(* PLC project Standard Funtion Blocks, Beremiz Additional Function Blocks Library 1.0, author Laurent Bessard *)
(* stored: creationDateTime 2013-09-09T09:56:11, modificationDateTime 2013-09-10T22:45:31 *)

(* pluse out *)
FUNCTION_BLOCK StepperDriver
  VAR_INPUT
    CH : USINT;  (* 输出通道,范围由控制器决定,1-n *)
    MaxSpeed : UDINT;  (* 设定最高速度,单位Hz *)
    Acceleration : UDINT;  (* 设定最高加减速,单位Hz *)
    StepPinPolarity : BOOL;  (* 脉冲输出极性设定 *)
    DirectionPolarity : BOOL;  (* 方向输出极性设定 *)
    TargetAbs : DINT;  (* 绝对目标位置设定 *)
    TargetRel : DINT;  (* 相对目标位置设定 *)
    TargetSet : USINT;  (* 目标位置设定,1=绝对位置,2=相对位置,其它=不修改 *)
    Position : DINT;  (* 当前位置设定 *)
    PositionSet : BOOL;  (* 当前位置设定,1有效 *)
    Run : BOOL;  (* 1=运行,0=停止 *)
  END_VAR
  VAR_OUTPUT
    Running : BOOL;  (* 运行状态,1=正在运行,0=停止 *)
    End : BOOL;  (* 1=到达指定位置,0=未到达指定位置,进入运行状态时清零 *)
    CurrentPosition : DINT;  (* 当前位置 *)
  END_VAR

                        
        {{

  setStepper(GetFbVar(CH),GetFbVar(MAXSPEED),GetFbVar(ACCELERATION),GetFbVar(STEPPINPOLARITY),GetFbVar(DIRECTIONPOLARITY),GetFbVar(TARGETABS),GetFbVar(TARGETREL),GetFbVar(TARGETSET),GetFbVar(POSITION),GetFbVar(POSITIONSET));
  SetFbVar(CURRENTPOSITION,getStepperPosition(GetFbVar(CH)));

}}

                    
END_FUNCTION_BLOCK
